// TIA Portal V17 export
// export: Created 2025-03-07T09:17:35.5301543Z, ExportSetting WithDefaults, DisplayName Totally Integrated Automation Portal, DisplayVersion V17 Update 8, DisplayName TIA Portal Openness, DisplayVersion V17 Update 8, DisplayName TIA Portal Version Control Interface, DisplayVersion V17, DisplayName SINAMICS Startdrive Advanced, DisplayVersion V17 SP2, DisplayName SINAMICS Startdrive G110M, G120, G120C, G120D, G120P, G115D, DisplayVersion V17 SP2, DisplayName SINAMICS Startdrive G130, G150, S120, S150, SINAMICS MV, S210, DisplayVersion V17 SP2, DisplayName STEP 7 Professional, DisplayVersion V17 Update 8, DisplayName SINUMERIK ONE STEP 7 Toolbox, DisplayVersion V17 Update 12, DisplayName SINUMERIK 840D sl STEP 7 Toolbox, DisplayVersion V17 Update 12, DisplayName STEP 7 Safety, DisplayVersion V17 Update 6, DisplayName WinCC Advanced, DisplayVersion V17 Update 8
DATA_BLOCK "DB428_OPERATOR_HELP"   // DB428
{ S7_Optimized_Access := 'FALSE' }
VERSION : 1.0
// stored: AutoNumber false, DBAccessibleFromOPCUA true, DBAccessibleFromWebserver true, IsOnlyStoredInLoadMemory false, IsWriteProtectedInAS false
   VAR RETAIN
      HELP_OPERATOR_0 : Bool;   // EMPTY
      HELP_OPERATOR_1 : Bool;   // EMPTY
      HELP_OPERATOR_2 : Bool;   // SPINDLE, POWER MODULE NOT READY
      HELP_OPERATOR_3 : Bool;   // AXIS X, POWER MODULE NOT READY
      HELP_OPERATOR_4 : Bool;   // AXIS Y, POWER MODULE NOT READY
      HELP_OPERATOR_5 : Bool;   // AXIS Z, POWER MODULE NOT READY
      HELP_OPERATOR_6 : Bool;   // AXIS Q, POWER MODULE NOT READY
      HELP_OPERATOR_7 : Bool;   // AXIS A, POWER MODULE NOT READY
      HELP_OPERATOR_8 : Bool;   // AXIS B, POWER MODULE NOT READY
      HELP_OPERATOR_9 : Bool;   // AXIS W, POWER MODULE NOT READY
      HELP_OPERATOR_10 : Bool;   // AXIS E, POWER MODULE NOT READY
      HELP_OPERATOR_11 : Bool;   // AXIS U, POWER MODULE NOT READY
      HELP_OPERATOR_12 : Bool;   // AXIS V, POWER MODULE NOT READY
      HELP_OPERATOR_13 : Bool;   // AXIS ROLLER, POWER MODULE NOT READY
      HELP_OPERATOR_14 : Bool;   // AXIS C, POWER MODULE NOT READY
      HELP_OPERATOR_15 : Bool;   // AXIS DR, POWER MODULE NOT READY
      HELP_OPERATOR_16 : Bool;
      HELP_OPERATOR_17 : Bool;
      HELP_OPERATOR_18 : Bool;
      HELP_OPERATOR_19 : Bool;
      HELP_OPERATOR_20 : Bool;
      HELP_OPERATOR_21 : Bool;
      HELP_OPERATOR_22 : Bool;
      HELP_OPERATOR_23 : Bool;
      HELP_OPERATOR_24 : Bool;
      HELP_OPERATOR_25 : Bool;   // SP11, SPEED NOT 0
      HELP_OPERATOR_26 : Bool;   // SP12, SPEED NOT 0
      HELP_OPERATOR_27 : Bool;   // SP13, SPEED NOT 0
      HELP_OPERATOR_28 : Bool;   // SP14, SPEED NOT 0
      HELP_OPERATOR_29 : Bool;
      HELP_OPERATOR_30 : Bool;
      HELP_OPERATOR_31 : Bool;
      HELP_OPERATOR_32 : Bool;
      HELP_OPERATOR_33 : Bool;   // SP21, SPEED NOT 0
      HELP_OPERATOR_34 : Bool;   // SP22, SPEED NOT 0
      HELP_OPERATOR_35 : Bool;   // SP23, SPEED NOT 0
      HELP_OPERATOR_36 : Bool;   // SP24, SPEED NOT 0
      HELP_OPERATOR_37 : Bool;
      HELP_OPERATOR_38 : Bool;   // RETURN AXIS E10 TO HOME POSITION
      HELP_OPERATOR_39 : Bool;   // RETURN AXIS X13 TO HOME POSITION
      HELP_OPERATOR_40 : Bool;   // RETURN AXIS W11 TO HOME POSITION
      HELP_OPERATOR_41 : Bool;   // RETURN AXIS Z13 TO HOME POSITION
      HELP_OPERATOR_42 : Bool;   // RETURN AXIS E20 TO HOME POSITION
      HELP_OPERATOR_43 : Bool;   // RETURN AXIS C22 TO HOME POSITION
      HELP_OPERATOR_44 : Bool;   // RETURN AXIS X23 TO HOME POSITION
      HELP_OPERATOR_45 : Bool;   // RETURN AXIS W21 TO HOME POSITION
      HELP_OPERATOR_46 : Bool;   // RETURN AXIS Z23 TO HOME POSITION
      HELP_OPERATOR_47 : Bool;   // RETURN AXIS C31 TO HOME POSITION
      HELP_OPERATOR_48 : Bool;
      HELP_OPERATOR_49 : Bool;   // RETURN AXIS X21 TO HOME POSITION
      HELP_OPERATOR_50 : Bool;   // RETURN AXIS Y21 TO HOME POSITION
      HELP_OPERATOR_51 : Bool;   // RETURN AXIS Z21 TO HOME POSITION
      HELP_OPERATOR_52 : Bool;   // RETURN AXIS Z22 TO HOME POSITION
      HELP_OPERATOR_53 : Bool;   // RETURN AXIS Z23 TO HOME POSITION
      HELP_OPERATOR_54 : Bool;   // RETURN AXIS Q21 TO HOME POSITION
      HELP_OPERATOR_55 : Bool;
      HELP_OPERATOR_56 : Bool;
      HELP_OPERATOR_57 : Bool;   // RETURN AXIS B TO HOME POSITION
      HELP_OPERATOR_58 : Bool;   // RETURN AXIS W TO HOME POSITION
      HELP_OPERATOR_59 : Bool;   // RETURN AXIS E TO HOME POSITION
      HELP_OPERATOR_60 : Bool;
      HELP_OPERATOR_61 : Bool;   // RETURN AXIS ROLLER TO HOME POSITION
      HELP_OPERATOR_62 : Bool;   // RETURN AXIS A11 TO HOME POSITION
      HELP_OPERATOR_63 : Bool;   // RETURN AXIS A12 TO HOME POSITION
      HELP_OPERATOR_64 : Bool;   // RETURN AXIS A13 TO HOME POSITION
      HELP_OPERATOR_65 : Bool;   // RETURN AXIS V11 TO HOME POSITION
      HELP_OPERATOR_66 : Bool;   // RETURN AXIS V12 TO HOME POSITION
      HELP_OPERATOR_67 : Bool;   // RETURN AXIS U11 TO HOME POSITION
      HELP_OPERATOR_68 : Bool;   // RETURN AXIS U12 TO HOME POSITION
      HELP_OPERATOR_69 : Bool;   // RETURN AXIS W11 TO HOME POSITION
      HELP_OPERATOR_70 : Bool;   // RETURN AXIS C TO HOME POSITION
      HELP_OPERATOR_71 : Bool;
      HELP_OPERATOR_72 : Bool;   // RETURN AXIS A21 TO HOME POSITION
      HELP_OPERATOR_73 : Bool;   // RETURN AXIS A22 TO HOME POSITION
      HELP_OPERATOR_74 : Bool;   // RETURN AXIS V21 TO HOME POSITION
      HELP_OPERATOR_75 : Bool;
      HELP_OPERATOR_76 : Bool;   // RETURN AXIS U21 TO HOME POSITION
      HELP_OPERATOR_77 : Bool;
      HELP_OPERATOR_78 : Bool;
      HELP_OPERATOR_79 : Bool;   // RETURN AXIS DR1 TO HOME POSITION
      HELP_OPERATOR_80 : Bool;   // RETURN AXIS DR2 TO HOME POSITION
      HELP_OPERATOR_81 : Bool;
      HELP_OPERATOR_82 : Bool;
      HELP_OPERATOR_83 : Bool;   // RETURN AXIS E10 TO OUT OF COLLISION POSITION
      HELP_OPERATOR_84 : Bool;   // RETURN AXIS X13 TO OUT OF COLLISION POSITION
      HELP_OPERATOR_85 : Bool;   // RETURN AXIS W11 TO OUT OF COLLISION POSITION
      HELP_OPERATOR_86 : Bool;   // RETURN AXIS Z13 TO OUT OF COLLISION POSITION
      HELP_OPERATOR_87 : Bool;   // RETURN AXIS E20 TO OUT OF COLLISION POSITION
      HELP_OPERATOR_88 : Bool;   // RETURN AXIS C22 TO OUT OF COLLISION POSITION
      HELP_OPERATOR_89 : Bool;   // RETURN AXIS X23 TO OUT OF COLLISION POSITION
      HELP_OPERATOR_90 : Bool;   // RETURN AXIS W21 TO OUT OF COLLISION POSITION
      HELP_OPERATOR_91 : Bool;   // RETURN AXIS Z23 TO OUT OF COLLISION POSITION
      HELP_OPERATOR_92 : Bool;   // RETURN AXIS C31 TO OUT OF COLLISION POSITION
      HELP_OPERATOR_93 : Bool;   // RETURN AXIS Z23 TO OUT OF COLLISION POSITION
      HELP_OPERATOR_94 : Bool;   // RETURN AXIS Q21 TO OUT OF COLLISION POSITION
      HELP_OPERATOR_95 : Bool;   // RETURN AXIS B TO OUT OF COLLISION POSITION
      HELP_OPERATOR_96 : Bool;   // RETURN AXIS W TO OUT OF COLLISION POSITION
      HELP_OPERATOR_97 : Bool;   // RETURN AXIS E TO OUT OF COLLISION POSITION
      HELP_OPERATOR_98 : Bool;
      HELP_OPERATOR_99 : Bool;   // RETURN AXIS ROLLER TO OUT OF COLLISION POSITION
      HELP_OPERATOR_100 : Bool;   // RETURN AXIS A11 TO OUT OF COLLISION POSITION
      HELP_OPERATOR_101 : Bool;   // RETURN AXIS A12 TO OUT OF COLLISION POSITION
      HELP_OPERATOR_102 : Bool;   // RETURN AXIS A13 TO OUT OF COLLISION POSITION
      HELP_OPERATOR_103 : Bool;   // RETURN AXIS V11 TO OUT OF COLLISION POSITION
      HELP_OPERATOR_104 : Bool;   // RETURN AXIS V12 TO OUT OF COLLISION POSITION
      HELP_OPERATOR_105 : Bool;   // RETURN AXIS U11 TO OUT OF COLLISION POSITION
      HELP_OPERATOR_106 : Bool;   // RETURN AXIS U12 TO OUT OF COLLISION POSITION
      HELP_OPERATOR_107 : Bool;   // RETURN AXIS W11 TO OUT OF COLLISION POSITION
      HELP_OPERATOR_108 : Bool;   // RETURN AXIS C TO OUT OF COLLISION POSITION
      HELP_OPERATOR_109 : Bool;
      HELP_OPERATOR_110 : Bool;   // RETURN AXIS A21 TO OUT OF COLLISION POSITION
      HELP_OPERATOR_111 : Bool;   // RETURN AXIS A22 TO OUT OF COLLISION POSITION
      HELP_OPERATOR_112 : Bool;   // RETURN AXIS V21 TO OUT OF COLLISION POSITION
      HELP_OPERATOR_113 : Bool;
      HELP_OPERATOR_114 : Bool;   // RETURN AXIS U21 TO OUT OF COLLISION POSITION
      HELP_OPERATOR_115 : Bool;
      HELP_OPERATOR_116 : Bool;   // RETURN AXIS DR1 TO OUT OF COLLISION POSITION
      HELP_OPERATOR_117 : Bool;   // RETURN AXIS DR2 TO OUT OF COLLISION POSITION
      HELP_OPERATOR_118 : Bool;
      HELP_OPERATOR_119 : Bool;   // AXIS B NOT IN -180º
      HELP_OPERATOR_120 : Bool;   // AXIS B NOT IN 0º
      HELP_OPERATOR_121 : Bool;   // ROTATE AXIS B TO ANY INDEXING POSITION
      HELP_OPERATOR_122 : Bool;
      HELP_OPERATOR_123 : Bool;
      HELP_OPERATOR_124 : Bool;   // AXIS NOT IN 90º
      HELP_OPERATOR_125 : Bool;   // AXIS NOT IN -90º
      HELP_OPERATOR_126 : Bool;
      HELP_OPERATOR_127 : Bool;
      HELP_OPERATOR_128 : Bool;   // ROTATE AXIS E TO 0º
      HELP_OPERATOR_129 : Bool;   // ROTATE AXIS E TO 180º
      HELP_OPERATOR_130 : Bool;
      HELP_OPERATOR_131 : Bool;
      HELP_OPERATOR_132 : Bool;   // ADVANCE AXIS A
      HELP_OPERATOR_133 : Bool;   // RETURN AXIS A
      HELP_OPERATOR_134 : Bool;   // MOVE AXIS A TO LOAD UNLOAD POSITION
      HELP_OPERATOR_135 : Bool;
      HELP_OPERATOR_136 : Bool;   // ADVANCE AXIS U
      HELP_OPERATOR_137 : Bool;   // RETURN AXIS U
      HELP_OPERATOR_138 : Bool;
      HELP_OPERATOR_139 : Bool;   // RETURN AXIS Q TO POSITION
      HELP_OPERATOR_140 : Bool;
      HELP_OPERATOR_141 : Bool;   // CHOOSE AXES TO ALIGN
      HELP_OPERATOR_142 : Bool;
      HELP_OPERATOR_143 : Bool;
      HELP_OPERATOR_144 : Bool;
      HELP_OPERATOR_145 : Bool;   // ADVANCE AXIS W11
      HELP_OPERATOR_146 : Bool;   // RETURN AXIS W11
      HELP_OPERATOR_147 : Bool;
      HELP_OPERATOR_148 : Bool;
      HELP_OPERATOR_149 : Bool;
      HELP_OPERATOR_150 : Bool;   // RETURN UNIT 01 TO HOME POSITION
      HELP_OPERATOR_151 : Bool;   // RETURN UNIT 02 TO HOME POSITION
      HELP_OPERATOR_152 : Bool;   // RETURN UNIT 03 TO HOME POSITION
      HELP_OPERATOR_153 : Bool;   // RETURN UNIT 04 TO HOME POSITION
      HELP_OPERATOR_154 : Bool;   // RETURN UNIT 05 TO HOME POSITION
      HELP_OPERATOR_155 : Bool;   // RETURN UNIT 06 TO HOME POSITION
      HELP_OPERATOR_156 : Bool;   // RETURN UNIT 07 TO HOME POSITION
      HELP_OPERATOR_157 : Bool;   // RETURN UNIT 08 TO HOME POSITION
      HELP_OPERATOR_158 : Bool;   // RETURN UNIT 09 TO HOME POSITION
      HELP_OPERATOR_159 : Bool;   // RETURN UNIT 10 TO HOME POSITION
      HELP_OPERATOR_160 : Bool;
      HELP_OPERATOR_161 : Bool;
      HELP_OPERATOR_162 : Bool;   // UNIT 01 IN HOME POSITION
      HELP_OPERATOR_163 : Bool;   // UNIT 02 IN HOME POSITION
      HELP_OPERATOR_164 : Bool;   // UNIT 03 IN HOME POSITION
      HELP_OPERATOR_165 : Bool;   // UNIT 04 IN HOME POSITION
      HELP_OPERATOR_166 : Bool;   // UNIT 5 IN HOME POSITION
      HELP_OPERATOR_167 : Bool;   // UNIT 6 IN HOME POSITION
      HELP_OPERATOR_168 : Bool;   // UNIT 7 IN HOME POSITION
      HELP_OPERATOR_169 : Bool;   // UNIT 8 IN HOME POSITION
      HELP_OPERATOR_170 : Bool;   // UNIT 9 IN HOME POSITION
      HELP_OPERATOR_171 : Bool;   // UNIT 10 IN HOME POSITION
      HELP_OPERATOR_172 : Bool;
      HELP_OPERATOR_173 : Bool;
      HELP_OPERATOR_174 : Bool;   // UNIT 01R SPINDLES NOT STOPPED
      HELP_OPERATOR_175 : Bool;   // UNIT 01L SPINDLES NOT STOPPED
      HELP_OPERATOR_176 : Bool;
      HELP_OPERATOR_177 : Bool;
      HELP_OPERATOR_178 : Bool;   // TOOLS IN MAGAZINE 01R NOT OK
      HELP_OPERATOR_179 : Bool;   // TOOLS IN MAGAZINE 01L NOT OK
      HELP_OPERATOR_180 : Bool;
      HELP_OPERATOR_181 : Bool;
      HELP_OPERATOR_182 : Bool;   // RETURN MACHINE TO HOME POSITION
      HELP_OPERATOR_183 : Bool;   // MACHINE IN HOME POSITION
      HELP_OPERATOR_184 : Bool;   // RETURN PART HANDLING DEVICE TO HOME POSITION
      HELP_OPERATOR_185 : Bool;   // PART HANDLING DEVICE IN HOME POSITION
      HELP_OPERATOR_186 : Bool;   // ADVANCE PHD TO LOAD UNLOAD POS FIXTURE
      HELP_OPERATOR_187 : Bool;
      HELP_OPERATOR_188 : Bool;
      HELP_OPERATOR_189 : Bool;
      HELP_OPERATOR_190 : Bool;   // NO PART AT FEED
      HELP_OPERATOR_191 : Bool;   // PARTS DELIVERY OCCUPIED
      HELP_OPERATOR_192 : Bool;
      HELP_OPERATOR_193 : Bool;
      HELP_OPERATOR_194 : Bool;
      HELP_OPERATOR_195 : Bool;
      HELP_OPERATOR_196 : Bool;
      HELP_OPERATOR_197 : Bool;
      HELP_OPERATOR_198 : Bool;
      HELP_OPERATOR_199 : Bool;
      HELP_OPERATOR_200 : Bool;   // SELECT MANUAL MODE
      HELP_OPERATOR_201 : Bool;   // SELECT JOG MODE
      HELP_OPERATOR_202 : Bool;   // SELECT SEMIAUTOMATIC MODE
      HELP_OPERATOR_203 : Bool;   // SELECT TOOL CHANGE MODE
      HELP_OPERATOR_204 : Bool;   // SELECT AUTOMATIC MODE
      HELP_OPERATOR_205 : Bool;   // SELECT INCREMENTAL MODE
      HELP_OPERATOR_206 : Bool;   // SELECT AUTO. OR SEMIAUTO. OR SINGLE MODE
      HELP_OPERATOR_207 : Bool;   // SELECT CALIBRATION CYCLE
      HELP_OPERATOR_208 : Bool;   // SELECT MEASUREMENT CYCLE
      HELP_OPERATOR_209 : Bool;
      HELP_OPERATOR_210 : Bool;
      HELP_OPERATOR_211 : Bool;
      HELP_OPERATOR_212 : Bool;
      HELP_OPERATOR_213 : Bool;
      HELP_OPERATOR_214 : Bool;
      HELP_OPERATOR_215 : Bool;   // UNSELECT REFERENCE MODE
      HELP_OPERATOR_216 : Bool;   // UNSELECT STEP BY STEP MODE
      HELP_OPERATOR_217 : Bool;   // UNSELECT MANUAL LOADING CYCLE
      HELP_OPERATOR_218 : Bool;   // UNSELECT MDA MODE
      HELP_OPERATOR_219 : Bool;   // UNSELECT RUN-OUT CYCLE
      HELP_OPERATOR_220 : Bool;   // UNSELECT DRY CYCLE
      HELP_OPERATOR_221 : Bool;   // UNSELECT GANTRY TEST CYCLE
      HELP_OPERATOR_222 : Bool;   // UNSELECT ROBOT DRY CYCLE
      HELP_OPERATOR_223 : Bool;   // UNSELECT SINGLE CYCLE
      HELP_OPERATOR_224 : Bool;   // UNSELECT CALIBRATION CYCLE
      HELP_OPERATOR_225 : Bool;
      HELP_OPERATOR_226 : Bool;
      HELP_OPERATOR_227 : Bool;
      HELP_OPERATOR_228 : Bool;
      HELP_OPERATOR_229 : Bool;
      HELP_OPERATOR_230 : Bool;   // ENABLE BA1 MODE
      HELP_OPERATOR_231 : Bool;   // ENABLE BA1 OR BA3 MODE
      HELP_OPERATOR_232 : Bool;   // ENABLE BA2 MODE OR CLOSE SAFETY DOORS
      HELP_OPERATOR_233 : Bool;
      HELP_OPERATOR_234 : Bool;
      HELP_OPERATOR_235 : Bool;
      HELP_OPERATOR_236 : Bool;   // SELECT POWDER PLC AUTO MODE
      HELP_OPERATOR_237 : Bool;
      HELP_OPERATOR_238 : Bool;
      HELP_OPERATOR_239 : Bool;
      HELP_OPERATOR_240 : Bool;
      HELP_OPERATOR_241 : Bool;
      HELP_OPERATOR_242 : Bool;
      HELP_OPERATOR_243 : Bool;
      HELP_OPERATOR_244 : Bool;
      HELP_OPERATOR_245 : Bool;
      HELP_OPERATOR_246 : Bool;
      HELP_OPERATOR_247 : Bool;
      HELP_OPERATOR_248 : Bool;
      HELP_OPERATOR_249 : Bool;
      HELP_OPERATOR_250 : Bool;   // OVERRIDE 0
      HELP_OPERATOR_251 : Bool;
      HELP_OPERATOR_252 : Bool;   // EMPTY THE MACHINE
      HELP_OPERATOR_253 : Bool;   // CLEAN GUIDES CYCLE REQUIRED
      HELP_OPERATOR_254 : Bool;   // DISABLE SAVE ENERGY
      HELP_OPERATOR_255 : Bool;   // EMPTY THE CELL
      HELP_OPERATOR_256 : Bool;   // SELECT MANUAL LOADING SELECTOR BUTTON
      HELP_OPERATOR_257 : Bool;
      HELP_OPERATOR_258 : Bool;   // RFID DATA CARRIER CODE MISSING
      HELP_OPERATOR_259 : Bool;   // READING IN PROCESS
      HELP_OPERATOR_260 : Bool;   // WRITING NOT IN PROCESS
      HELP_OPERATOR_261 : Bool;
      HELP_OPERATOR_262 : Bool;
      HELP_OPERATOR_263 : Bool;   // ACKNOWLEDGE QUALITY CHECK
      HELP_OPERATOR_264 : Bool;   // ACKNOWLEDGE ON DEMAND QUALITY CHECK
      HELP_OPERATOR_265 : Bool;   // ACKNOWLEDGE TOOL CHANGED QUALITY CHECK
      HELP_OPERATOR_266 : Bool;   // ACKNOWLEDGE PART TYPE CHANGED QUALITY CHECK
      HELP_OPERATOR_267 : Bool;   // ACKNOWLEDGE FIRST PART QUALITY CHECK
      HELP_OPERATOR_268 : Bool;   // ACKNOWLEDGE CYCLE INTERRUPTED QUALITY CHECK
      HELP_OPERATOR_269 : Bool;   // STOP ACTUAL CYCLE
      HELP_OPERATOR_270 : Bool;   // MACHINE SEQUENCE IN PROGRESS
      HELP_OPERATOR_271 : Bool;   // TEST STOP SEQUENCE IN PROGRESS
      HELP_OPERATOR_272 : Bool;   // SEQUENCE IN PROGRESS
      HELP_OPERATOR_273 : Bool;
      HELP_OPERATOR_274 : Bool;   // LASER FAULT
      HELP_OPERATOR_275 : Bool;   // LASER IS NOT ACTIVE
      HELP_OPERATOR_276 : Bool;   // LASER DEVICE IS NOT READY
      HELP_OPERATOR_277 : Bool;   // LASER EXTERNAL CONTROL IS NOT READY
      HELP_OPERATOR_278 : Bool;   // LASER POINTER FAULT
      HELP_OPERATOR_279 : Bool;
      HELP_OPERATOR_280 : Bool;   // START POWDER UNIT 01
      HELP_OPERATOR_281 : Bool;   // START POWDER UNIT 02
      HELP_OPERATOR_282 : Bool;
      HELP_OPERATOR_283 : Bool;
      HELP_OPERATOR_284 : Bool;
      HELP_OPERATOR_285 : Bool;
      HELP_OPERATOR_286 : Bool;
      HELP_OPERATOR_287 : Bool;
      HELP_OPERATOR_288 : Bool;
      HELP_OPERATOR_289 : Bool;
      HELP_OPERATOR_290 : Bool;   // ACTION ALREADY DONE
      HELP_OPERATOR_291 : Bool;
      HELP_OPERATOR_292 : Bool;
      HELP_OPERATOR_293 : Bool;
      HELP_OPERATOR_294 : Bool;   // JOG MINUS IS NOT ALLOWED
      HELP_OPERATOR_295 : Bool;   // JOG PLUS IS NOT ALLOWED
      HELP_OPERATOR_296 : Bool;
      HELP_OPERATOR_297 : Bool;
      HELP_OPERATOR_298 : Bool;
      HELP_OPERATOR_299 : Bool;
      HELP_OPERATOR_300 : Bool;   // SAFETY GATES NOT CLOSED AND LOCKED
      HELP_OPERATOR_301 : Bool;   // CLOSE AND LOCK MACHINING STATION SAFETY DOOR
      HELP_OPERATOR_302 : Bool;   // OPEN AND UNLOCK MACHINING STATION SAFETY DOOR
      HELP_OPERATOR_303 : Bool;   // CLOSE AND LOCK LOAD/ UNLOAD STATION SAFETY DOOR
      HELP_OPERATOR_304 : Bool;   // OPEN AND UNLOCK LOAD UNLOAD STATION SAFETY DOOR
      HELP_OPERATOR_305 : Bool;   // CLOSE AND LOCK PART HANDLING DEVICE SAFETY DOOR
      HELP_OPERATOR_306 : Bool;   // OPEN AND UNLOCK PART HANDLING DEVICE SAFETY DOOR
      HELP_OPERATOR_307 : Bool;
      HELP_OPERATOR_308 : Bool;   // BIMANUAL NOT PRESSED
      HELP_OPERATOR_309 : Bool;
      HELP_OPERATOR_310 : Bool;
      HELP_OPERATOR_311 : Bool;   // CLOSE AND LOCK TOOL MAGAZINE 01 R SAFETY DOOR
      HELP_OPERATOR_312 : Bool;   // OPEN AND UNLOCK TOOL MAGAZINE 01R SAFETY DOOR
      HELP_OPERATOR_313 : Bool;   // CLOSE AND LOCK TOOL MAGAZINE 01L SAFETY DOOR
      HELP_OPERATOR_314 : Bool;   // OPEN AND UNLOCK TOOL MAGAZINE 01L SAFETY DOOR
      HELP_OPERATOR_315 : Bool;
      HELP_OPERATOR_316 : Bool;
      HELP_OPERATOR_317 : Bool;   // CLOSE AND LOCK UNIT 01 R SAFETY DOOR
      HELP_OPERATOR_318 : Bool;   // OPEN AND UNLOCK UNIT 01R SAFETY DOOR
      HELP_OPERATOR_319 : Bool;   // CLOSE AND LOCK UNIT 01L SAFETY DOOR
      HELP_OPERATOR_320 : Bool;   // OPEN AND UNLOCK UNIT 01L SAFETY DOOR
      HELP_OPERATOR_321 : Bool;
      HELP_OPERATOR_322 : Bool;
      HELP_OPERATOR_323 : Bool;
      HELP_OPERATOR_324 : Bool;
      HELP_OPERATOR_325 : Bool;   // CLOSE AND LOCK MAINTENANCE PLATFORM SAFETY DOOR
      HELP_OPERATOR_326 : Bool;   // OPEN AND UNLOCK MAINTENANCE PLATFORM SAFETY DOOR
      HELP_OPERATOR_327 : Bool;
      HELP_OPERATOR_328 : Bool;
      HELP_OPERATOR_329 : Bool;   // CLOSE AND LOCK CHIP CRUSHER SAFETY DOOR
      HELP_OPERATOR_330 : Bool;   // OPEN AND UNLOCK CHIP CRUSHER SAFETY DOOR
      HELP_OPERATOR_331 : Bool;
      HELP_OPERATOR_332 : Bool;
      HELP_OPERATOR_333 : Bool;   // CLOSE MACHINING STATION SAFETY DOOR
      HELP_OPERATOR_334 : Bool;   // CLOSE LOAD UNLOAD STATION SAFETY DOOR
      HELP_OPERATOR_335 : Bool;   // CLOSE PART HANDLING DEVICE SAFETY DOOR
      HELP_OPERATOR_336 : Bool;
      HELP_OPERATOR_337 : Bool;
      HELP_OPERATOR_338 : Bool;   // CLOSE TOOL MAGAZINE 01R SAFETY DOOR
      HELP_OPERATOR_339 : Bool;   // CLOSE TOOL MAGAZINE 01L SAFETY DOOR
      HELP_OPERATOR_340 : Bool;
      HELP_OPERATOR_341 : Bool;   // CLOSE UNIT 01R SAFETY DOOR
      HELP_OPERATOR_342 : Bool;   // CLOSE UNIT 01L SAFETY DOOR
      HELP_OPERATOR_343 : Bool;
      HELP_OPERATOR_344 : Bool;
      HELP_OPERATOR_345 : Bool;   // CLOSE MAINTENANCE PLATFORM SAFETY DOOR
      HELP_OPERATOR_346 : Bool;
      HELP_OPERATOR_347 : Bool;   // CLOSE CHIP CRUSHER SAFETY DOOR
      HELP_OPERATOR_348 : Bool;
      HELP_OPERATOR_349 : Bool;
      HELP_OPERATOR_350 : Bool;   // PART TYPE 1 SELECTED
      HELP_OPERATOR_351 : Bool;   // PART TYPE 2 SELECTED
      HELP_OPERATOR_352 : Bool;   // PART TYPE 3 SELECTED
      HELP_OPERATOR_353 : Bool;   // PART TYPE 4 SELECTED
      HELP_OPERATOR_354 : Bool;   // PART TYPE 5 SELECTED
      HELP_OPERATOR_355 : Bool;   // PART TYPE 6 SELECTED
      HELP_OPERATOR_356 : Bool;   // PART TYPE 7 SELECTED
      HELP_OPERATOR_357 : Bool;   // PART TYPE 8 SELECTED
      HELP_OPERATOR_358 : Bool;   // PART TYPE 9 SELECTED
      HELP_OPERATOR_359 : Bool;   // PART TYPE 10 SELECTED
      HELP_OPERATOR_360 : Bool;   // PART TYPE 11 SELECTED
      HELP_OPERATOR_361 : Bool;   // PART TYPE 12 SELECTED
      HELP_OPERATOR_362 : Bool;   // PART TYPE 13 SELECTED
      HELP_OPERATOR_363 : Bool;   // PART TYPE 14 SELECTED
      HELP_OPERATOR_364 : Bool;   // PART TYPE 15 SELECTED
      HELP_OPERATOR_365 : Bool;   // PART TYPE 16 SELECTED
      HELP_OPERATOR_366 : Bool;   // PART TYPE 17 SELECTED
      HELP_OPERATOR_367 : Bool;   // PART TYPE 18 SELECTED
      HELP_OPERATOR_368 : Bool;   // PART TYPE 19 SELECTED
      HELP_OPERATOR_369 : Bool;   // PART TYPE 20 SELECTED
      HELP_OPERATOR_370 : Bool;   // PART TYPE 21 SELECTED
      HELP_OPERATOR_371 : Bool;   // PART TYPE 22 SELECTED
      HELP_OPERATOR_372 : Bool;   // PART TYPE 23 SELECTED
      HELP_OPERATOR_373 : Bool;   // PART TYPE 24 SELECTED
      HELP_OPERATOR_374 : Bool;   // PART TYPE 25 SELECTED
      HELP_OPERATOR_375 : Bool;   // PART TYPE 26 SELECTED
      HELP_OPERATOR_376 : Bool;   // PART TYPE 27 SELECTED
      HELP_OPERATOR_377 : Bool;   // PART TYPE 28 SELECTED
      HELP_OPERATOR_378 : Bool;   // PART TYPE 29 SELECTED
      HELP_OPERATOR_379 : Bool;   // PART TYPE 30 SELECTED
      HELP_OPERATOR_380 : Bool;   // PART TYPE 31 SELECTED
      HELP_OPERATOR_381 : Bool;   // PART TYPE 32 SELECTED
      HELP_OPERATOR_382 : Bool;
      HELP_OPERATOR_383 : Bool;
      HELP_OPERATOR_384 : Bool;
      HELP_OPERATOR_385 : Bool;
      HELP_OPERATOR_386 : Bool;
      HELP_OPERATOR_387 : Bool;
      HELP_OPERATOR_388 : Bool;
      HELP_OPERATOR_389 : Bool;
      HELP_OPERATOR_390 : Bool;
      HELP_OPERATOR_391 : Bool;
      HELP_OPERATOR_392 : Bool;
      HELP_OPERATOR_393 : Bool;
      HELP_OPERATOR_394 : Bool;
      HELP_OPERATOR_395 : Bool;
      HELP_OPERATOR_396 : Bool;
      HELP_OPERATOR_397 : Bool;
      HELP_OPERATOR_398 : Bool;
      HELP_OPERATOR_399 : Bool;
      HELP_OPERATOR_400 : Bool;   // CONFIRM HARDWARE DISABLING
      HELP_OPERATOR_401 : Bool;
      HELP_OPERATOR_402 : Bool;   // PART A DISABLED
      HELP_OPERATOR_403 : Bool;   // PART B DISABLED
      HELP_OPERATOR_404 : Bool;   // PART C DISABLED
      HELP_OPERATOR_405 : Bool;   // PART D DISABLED
      HELP_OPERATOR_406 : Bool;
      HELP_OPERATOR_407 : Bool;
      HELP_OPERATOR_408 : Bool;
      HELP_OPERATOR_409 : Bool;
      HELP_OPERATOR_410 : Bool;   // FIXTURE 1 DISABLED
      HELP_OPERATOR_411 : Bool;   // FIXTURE 2 DISABLED
      HELP_OPERATOR_412 : Bool;
      HELP_OPERATOR_413 : Bool;
      HELP_OPERATOR_414 : Bool;   // UNIT 01 DISABLED
      HELP_OPERATOR_415 : Bool;   // UNIT 02 DISABLED
      HELP_OPERATOR_416 : Bool;   // UNIT 03 DISABLED
      HELP_OPERATOR_417 : Bool;
      HELP_OPERATOR_418 : Bool;
      HELP_OPERATOR_419 : Bool;   // ALL BK MIKRO 01R UNITS DISABLED
      HELP_OPERATOR_420 : Bool;   // ALL BK MIKRO 01L UNITS DISABLED
      HELP_OPERATOR_421 : Bool;
      HELP_OPERATOR_422 : Bool;
      HELP_OPERATOR_423 : Bool;
      HELP_OPERATOR_424 : Bool;   // LASER SOURCE DISABLED
      HELP_OPERATOR_425 : Bool;
      HELP_OPERATOR_426 : Bool;
      HELP_OPERATOR_427 : Bool;
      HELP_OPERATOR_428 : Bool;
      HELP_OPERATOR_429 : Bool;
      HELP_OPERATOR_430 : Bool;
      HELP_OPERATOR_431 : Bool;
      HELP_OPERATOR_432 : Bool;
      HELP_OPERATOR_433 : Bool;
      HELP_OPERATOR_434 : Bool;
      HELP_OPERATOR_435 : Bool;
      HELP_OPERATOR_436 : Bool;
      HELP_OPERATOR_437 : Bool;
      HELP_OPERATOR_438 : Bool;
      HELP_OPERATOR_439 : Bool;
      HELP_OPERATOR_440 : Bool;   // PHD ARM 1, PART PRESENT
      HELP_OPERATOR_441 : Bool;   // PHD ARM 2, PART PRESENT
      HELP_OPERATOR_442 : Bool;
      HELP_OPERATOR_443 : Bool;
      HELP_OPERATOR_444 : Bool;   // NO PART PRESENT
      HELP_OPERATOR_445 : Bool;   // NO MASTER PART PRESENT
      HELP_OPERATOR_446 : Bool;   // FIXTURE IN UNIT 01 CLADDING STATION NOT CLAMPED
      HELP_OPERATOR_447 : Bool;
      HELP_OPERATOR_448 : Bool;
      HELP_OPERATOR_449 : Bool;
      HELP_OPERATOR_450 : Bool;
      HELP_OPERATOR_451 : Bool;
      HELP_OPERATOR_452 : Bool;
      HELP_OPERATOR_453 : Bool;
      HELP_OPERATOR_454 : Bool;
      HELP_OPERATOR_455 : Bool;
      HELP_OPERATOR_456 : Bool;
      HELP_OPERATOR_457 : Bool;
      HELP_OPERATOR_458 : Bool;
      HELP_OPERATOR_459 : Bool;
      HELP_OPERATOR_460 : Bool;   // SP11, TOOL CLAMPING CLAMPED WITHOUT TOOL
      HELP_OPERATOR_461 : Bool;   // SP12, TOOL CLAMPING CLAMPED WITHOUT TOOL
      HELP_OPERATOR_462 : Bool;   // SP13, TOOL CLAMPING CLAMPED WITHOUT TOOL
      HELP_OPERATOR_463 : Bool;   // SP14, TOOL CLAMPING CLAMPED WITHOUT TOOL
      HELP_OPERATOR_464 : Bool;
      HELP_OPERATOR_465 : Bool;
      HELP_OPERATOR_466 : Bool;   // SP21, TOOL CLAMPING CLAMPED WITHOUT TOOL
      HELP_OPERATOR_467 : Bool;   // SP22, TOOL CLAMPING CLAMPED WITHOUT TOOL
      HELP_OPERATOR_468 : Bool;   // SP23, TOOL CLAMPING CLAMPED WITHOUT TOOL
      HELP_OPERATOR_469 : Bool;   // SP24, TOOL CLAMPING CLAMPED WITHOUT TOOL
      HELP_OPERATOR_470 : Bool;
      HELP_OPERATOR_471 : Bool;
      HELP_OPERATOR_472 : Bool;   // SP11, UNCLAMP TOOL CLAMPING
      HELP_OPERATOR_473 : Bool;   // SP12, UNCLAMP TOOL CLAMPING
      HELP_OPERATOR_474 : Bool;   // SP13, UNCLAMP TOOL CLAMPING
      HELP_OPERATOR_475 : Bool;   // SP14, UNCLAMP TOOL CLAMPING
      HELP_OPERATOR_476 : Bool;
      HELP_OPERATOR_477 : Bool;
      HELP_OPERATOR_478 : Bool;   // SP21, UNCLAMP TOOL CLAMPING
      HELP_OPERATOR_479 : Bool;   // SP22, UNCLAMP TOOL CLAMPING
      HELP_OPERATOR_480 : Bool;   // SP23, UNCLAMP TOOL CLAMPING
      HELP_OPERATOR_481 : Bool;   // SP24, UNCLAMP TOOL CLAMPING
      HELP_OPERATOR_482 : Bool;
      HELP_OPERATOR_483 : Bool;
      HELP_OPERATOR_484 : Bool;   // SP11, CLAMP TOOL CLAMPING
      HELP_OPERATOR_485 : Bool;   // SP12, CLAMP TOOL CLAMPING
      HELP_OPERATOR_486 : Bool;   // SP13, CLAMP TOOL CLAMPING
      HELP_OPERATOR_487 : Bool;   // SP14, CLAMP TOOL CLAMPING
      HELP_OPERATOR_488 : Bool;
      HELP_OPERATOR_489 : Bool;
      HELP_OPERATOR_490 : Bool;   // SP21, CLAMP TOOL CLAMPING
      HELP_OPERATOR_491 : Bool;   // SP22, CLAMP TOOL CLAMPING
      HELP_OPERATOR_492 : Bool;   // SP23, CLAMP TOOL CLAMPING
      HELP_OPERATOR_493 : Bool;   // SP24, CLAMP TOOL CLAMPING
      HELP_OPERATOR_494 : Bool;
      HELP_OPERATOR_495 : Bool;
      HELP_OPERATOR_496 : Bool;   // CLAMP WITH TOOL
      HELP_OPERATOR_497 : Bool;   // CLAMP TOOL CLAMPING
      HELP_OPERATOR_498 : Bool;
      HELP_OPERATOR_499 : Bool;   // MOVE TOOL FROM SP11 TO TOOL MAGAZINE 01R
      HELP_OPERATOR_500 : Bool;   // MOVE TOOL FROM SP12 TO TOOL MAGAZINE 01R
      HELP_OPERATOR_501 : Bool;   // MOVE TOOL FROM SP13 TO TOOL MAGAZINE 01R
      HELP_OPERATOR_502 : Bool;   // MOVE TOOL FROM SP14 TO TOOL MAGAZINE 01R
      HELP_OPERATOR_503 : Bool;
      HELP_OPERATOR_504 : Bool;
      HELP_OPERATOR_505 : Bool;   // MOVE TOOL FROM SP21 TO TOOL MAGAZINE 01L
      HELP_OPERATOR_506 : Bool;   // MOVE TOOL FROM SP22 TO TOOL MAGAZINE 01L
      HELP_OPERATOR_507 : Bool;   // MOVE TOOL FROM SP23 TO TOOL MAGAZINE 01L
      HELP_OPERATOR_508 : Bool;   // MOVE TOOL FROM SP24 TO TOOL MAGAZINE 01L
      HELP_OPERATOR_509 : Bool;
      HELP_OPERATOR_510 : Bool;
      HELP_OPERATOR_511 : Bool;   // SP11, ENABLE TOOL MONITORING
      HELP_OPERATOR_512 : Bool;   // SP12, ENABLE TOOL MONITORING
      HELP_OPERATOR_513 : Bool;   // SP13, ENABLE TOOL MONITORING
      HELP_OPERATOR_514 : Bool;   // SP14, ENABLE TOOL MONITORING
      HELP_OPERATOR_515 : Bool;
      HELP_OPERATOR_516 : Bool;
      HELP_OPERATOR_517 : Bool;   // SP21, ENABLE TOOL MONITORING
      HELP_OPERATOR_518 : Bool;   // SP22, ENABLE TOOL MONITORING
      HELP_OPERATOR_519 : Bool;   // SP23, ENABLE TOOL MONITORING
      HELP_OPERATOR_520 : Bool;   // SP24, ENABLE TOOL MONITORING
      HELP_OPERATOR_521 : Bool;
      HELP_OPERATOR_522 : Bool;
      HELP_OPERATOR_523 : Bool;   // BK MIKRO SP11 SEND TO HOME POS OR DISCONNECT CABLE
      HELP_OPERATOR_524 : Bool;   // BK MIKRO SP12 SEND TO HOME POS OR DISCONNECT CABLE
      HELP_OPERATOR_525 : Bool;   // BK MIKRO SP13 SEND TO HOME POS OR DISCONNECT CABLE
      HELP_OPERATOR_526 : Bool;   // BK MIKRO SP14 SEND TO HOME POS OR DISCONNECT CABLE
      HELP_OPERATOR_527 : Bool;
      HELP_OPERATOR_528 : Bool;
      HELP_OPERATOR_529 : Bool;   // BK MIKRO SP21 SEND TO HOME POS OR DISCONNECT CABLE
      HELP_OPERATOR_530 : Bool;   // BK MIKRO SP22 SEND TO HOME POS OR DISCONNECT CABLE
      HELP_OPERATOR_531 : Bool;   // BK MIKRO SP23 SEND TO HOME POS OR DISCONNECT CABLE
      HELP_OPERATOR_532 : Bool;   // BK MIKRO SP24 SEND TO HOME POS OR DISCONNECT CABLE
      HELP_OPERATOR_533 : Bool;
      HELP_OPERATOR_534 : Bool;
      HELP_OPERATOR_535 : Bool;   // MAIN OPERATOR PANEL, PRESS BUTTON CONTROL ON
      HELP_OPERATOR_536 : Bool;   // MAIN OPERATOR PANEL, PRESS BUTTON RESET
      HELP_OPERATOR_537 : Bool;   // REMOVE EMERGENCY STOPS, PRESS RESET FAULTS
      HELP_OPERATOR_538 : Bool;   // MACHINE STOP SERVICES DELAYED ENABLED
      HELP_OPERATOR_539 : Bool;
      HELP_OPERATOR_540 : Bool;
      HELP_OPERATOR_541 : Bool;   // SWITCH ON HYDRAULIC SYSTEM
      HELP_OPERATOR_542 : Bool;   // SWITCH ON PNEUMATIC SYSTEM
      HELP_OPERATOR_543 : Bool;   // LUBRICATION PRESSURES SWITCHES NOT BELOW 2 BARS
      HELP_OPERATOR_544 : Bool;   // MAIN CHIP CONVEYOR CONTAINER NOT PRESENT
      HELP_OPERATOR_545 : Bool;
      HELP_OPERATOR_546 : Bool;
      HELP_OPERATOR_547 : Bool;   // OPEN COOLANT VALVE
      HELP_OPERATOR_548 : Bool;   // SWITCH ON CHIP CRUSHER
      HELP_OPERATOR_549 : Bool;   // SWITCH OFF CHIP CRUSHER
      HELP_OPERATOR_550 : Bool;
      HELP_OPERATOR_551 : Bool;
      HELP_OPERATOR_552 : Bool;   // FILTER PAPER BAND HIGH LEVEL
      HELP_OPERATOR_553 : Bool;   // NOT READY
      HELP_OPERATOR_554 : Bool;   // LOW LEVEL
      HELP_OPERATOR_555 : Bool;   // NO PRESSURE AT INPUT
      HELP_OPERATOR_556 : Bool;   // FILTER CLOGGED
      HELP_OPERATOR_557 : Bool;
      HELP_OPERATOR_558 : Bool;
      HELP_OPERATOR_559 : Bool;   // FLUSH FILTER 01R NOT IN HOME POSITION
      HELP_OPERATOR_560 : Bool;   // FLUSH FILTER 01L NOT IN HOME POSITION
      HELP_OPERATOR_561 : Bool;
      HELP_OPERATOR_562 : Bool;
      HELP_OPERATOR_563 : Bool;
      HELP_OPERATOR_564 : Bool;
      HELP_OPERATOR_565 : Bool;   // SWITCH ON MQL PUMP
      HELP_OPERATOR_566 : Bool;
      HELP_OPERATOR_567 : Bool;   // SWITCH OFF MQL SP11
      HELP_OPERATOR_568 : Bool;   // SWITCH OFF MQL SP12
      HELP_OPERATOR_569 : Bool;   // SWITCH OFF MQL SP13
      HELP_OPERATOR_570 : Bool;   // SWITCH OFF MQL SP14
      HELP_OPERATOR_571 : Bool;
      HELP_OPERATOR_572 : Bool;
      HELP_OPERATOR_573 : Bool;   // SWITCH OFF MQL SP21
      HELP_OPERATOR_574 : Bool;   // SWITCH OFF MQL SP22
      HELP_OPERATOR_575 : Bool;   // SWITCH OFF MQL SP23
      HELP_OPERATOR_576 : Bool;   // SWITCH OFF MQL SP24
      HELP_OPERATOR_577 : Bool;
      HELP_OPERATOR_578 : Bool;
      HELP_OPERATOR_579 : Bool;
      HELP_OPERATOR_580 : Bool;
      HELP_OPERATOR_581 : Bool;
      HELP_OPERATOR_582 : Bool;
      HELP_OPERATOR_583 : Bool;
      HELP_OPERATOR_584 : Bool;
      HELP_OPERATOR_585 : Bool;
      HELP_OPERATOR_586 : Bool;
      HELP_OPERATOR_587 : Bool;
      HELP_OPERATOR_588 : Bool;
      HELP_OPERATOR_589 : Bool;
      HELP_OPERATOR_590 : Bool;   // CLAMP FIXTURE 1
      HELP_OPERATOR_591 : Bool;   // UNCLAMP FIXTURE 1
      HELP_OPERATOR_592 : Bool;   // CLAMP OR UNCLAMP FIXTURE 1
      HELP_OPERATOR_593 : Bool;   // FIXTURE 1, CLAMPED
      HELP_OPERATOR_594 : Bool;   // FIXTURE 1, UNCLAMPED
      HELP_OPERATOR_595 : Bool;   // SELECT PART TYPE FIXTURE 1
      HELP_OPERATOR_596 : Bool;   // FIXTURE 1 PART NOT OK
      HELP_OPERATOR_597 : Bool;   // CLAMPING SEQUENCE F1 IN PROGRESS
      HELP_OPERATOR_598 : Bool;
      HELP_OPERATOR_599 : Bool;   // CLAMP FIXTURE 2
      HELP_OPERATOR_600 : Bool;   // UNCLAMP FIXTURE 2
      HELP_OPERATOR_601 : Bool;   // CLAMP OR UNCLAMP FIXTURE 2
      HELP_OPERATOR_602 : Bool;   // FIXTURE 2, CLAMPED
      HELP_OPERATOR_603 : Bool;   // FIXTURE 2, UNCLAMPED
      HELP_OPERATOR_604 : Bool;   // SELECT PART TYPE FIXTURE 2
      HELP_OPERATOR_605 : Bool;   // FIXTURE 2 PART NOT OK
      HELP_OPERATOR_606 : Bool;   // CLAMPING SEQUENCE F2 IN PROGRESS
      HELP_OPERATOR_607 : Bool;
      HELP_OPERATOR_608 : Bool;   // CLAMP FIXTURE 3
      HELP_OPERATOR_609 : Bool;   // UNCLAMP FIXTURE 3
      HELP_OPERATOR_610 : Bool;   // CLAMP OR UNCLAMP FIXTURE 3
      HELP_OPERATOR_611 : Bool;   // FIXTURE 3, CLAMPED
      HELP_OPERATOR_612 : Bool;   // FIXTURE 3, UNCLAMPED
      HELP_OPERATOR_613 : Bool;   // SELECT PART TYPE FIXTURE 3
      HELP_OPERATOR_614 : Bool;   // FIXTURE 3 PART NOT OK
      HELP_OPERATOR_615 : Bool;   // CLAMPING SEQUENCE F3 IN PROGRESS
      HELP_OPERATOR_616 : Bool;
      HELP_OPERATOR_617 : Bool;   // CLAMP FIXTURE 4
      HELP_OPERATOR_618 : Bool;   // UNCLAMP FIXTURE 4
      HELP_OPERATOR_619 : Bool;   // CLAMP OR UNCLAMP FIXTURE 4
      HELP_OPERATOR_620 : Bool;   // FIXTURE 4, CLAMPED
      HELP_OPERATOR_621 : Bool;   // FIXTURE 4, UNCLAMPED
      HELP_OPERATOR_622 : Bool;   // SELECT PART TYPE FIXTURE 4
      HELP_OPERATOR_623 : Bool;   // FIXTURE 4 PART NOT OK
      HELP_OPERATOR_624 : Bool;   // CLAMPING SEQUENCE F4 IN PROGRESS
      HELP_OPERATOR_625 : Bool;
      HELP_OPERATOR_626 : Bool;   // LOCATE AXIAL LOCATOR
      HELP_OPERATOR_627 : Bool;   // LOCATE AXIAL LOCATOR CARRIER
      HELP_OPERATOR_628 : Bool;   // LOCATE RADIAL LOCATOR
      HELP_OPERATOR_629 : Bool;   // LOCATE RADIAL LOCATOR CARRIER
      HELP_OPERATOR_630 : Bool;   // CLAMP CLAMPING FLANGE
      HELP_OPERATOR_631 : Bool;   // ADVANCE TAILSTOCK
      HELP_OPERATOR_632 : Bool;   // LOCATE SHIFTING DEVICE
      HELP_OPERATOR_633 : Bool;   // BLOCK BLOCKING DEVICE
      HELP_OPERATOR_634 : Bool;   // CLAMP VIBRATION DAMPER
      HELP_OPERATOR_635 : Bool;   // CLAMP JAW CHUCK
      HELP_OPERATOR_636 : Bool;   // CLAMP CENTRAL JAWCHUCK
      HELP_OPERATOR_637 : Bool;   // CLAMP ROTARY JAW CHUCK
      HELP_OPERATOR_638 : Bool;   // ADVANCE REMOVABLE STOP
      HELP_OPERATOR_639 : Bool;
      HELP_OPERATOR_640 : Bool;
      HELP_OPERATOR_641 : Bool;
      HELP_OPERATOR_642 : Bool;   // CLAMP OR UNCLAMP FIXTURE IN UNIT 01 STATION 1
      HELP_OPERATOR_643 : Bool;   // CLAMP FIXTURE IN UNIT 1 STATION 3
      HELP_OPERATOR_644 : Bool;   // CLAMP FIXTURE IN UNIT 1 STATION 4
      HELP_OPERATOR_645 : Bool;   // CLAMP OR UNCLAMP FIXTURE IN UNIT 02 STATION 1
      HELP_OPERATOR_646 : Bool;   // CLAMP FIXTURE IN UNIT 2 STATION 2
      HELP_OPERATOR_647 : Bool;   // CLAMP FIXTURE IN UNIT 2 STATION 3
      HELP_OPERATOR_648 : Bool;   // CLAMP FIXTURE IN UNIT 2 STATION 4
      HELP_OPERATOR_649 : Bool;
      HELP_OPERATOR_650 : Bool;   // RETURN STATION 1 TO HOME POSITION
      HELP_OPERATOR_651 : Bool;   // RETURN STATION 2 TO HOME POSITION
      HELP_OPERATOR_652 : Bool;   // RETURN STATION 3 TO HOME POSITION
      HELP_OPERATOR_653 : Bool;   // RETURN STATION 4 TO HOME POSITION
      HELP_OPERATOR_654 : Bool;
      HELP_OPERATOR_655 : Bool;
      HELP_OPERATOR_656 : Bool;   // UNIT 01 ALL FIXTURES NOT CLAMPED
      HELP_OPERATOR_657 : Bool;   // UNIT 02 ALL FIXTURES NOT CLAMPED
      HELP_OPERATOR_658 : Bool;
      HELP_OPERATOR_659 : Bool;
      HELP_OPERATOR_660 : Bool;
      HELP_OPERATOR_661 : Bool;
      HELP_OPERATOR_662 : Bool;
      HELP_OPERATOR_663 : Bool;
      HELP_OPERATOR_664 : Bool;   // RETURN AXIAL LOCATOR
      HELP_OPERATOR_665 : Bool;   // RETURN AXIAL LOCATOR CARRIER
      HELP_OPERATOR_666 : Bool;   // RETURN RADIAL LOCATOR
      HELP_OPERATOR_667 : Bool;   // RETURN RADIAL LOCATOR CARRIER
      HELP_OPERATOR_668 : Bool;   // UNCLAMP CLAMPING FLANGE
      HELP_OPERATOR_669 : Bool;   // RETURN TAILSTOCK
      HELP_OPERATOR_670 : Bool;   // RETURN SHIFTING DEVICE
      HELP_OPERATOR_671 : Bool;   // UNBLOCK BLOCKING DEVICE
      HELP_OPERATOR_672 : Bool;   // UNCLAMP VIBRATION DAMPER
      HELP_OPERATOR_673 : Bool;   // UNCLAMP JAW CHUCK
      HELP_OPERATOR_674 : Bool;   // UNCLAMP CENTRAL JAWCHUCK
      HELP_OPERATOR_675 : Bool;   // UNCLAMP ROTARY JAW CHUCK
      HELP_OPERATOR_676 : Bool;   // RETURN REMOVABLE STOP
      HELP_OPERATOR_677 : Bool;
      HELP_OPERATOR_678 : Bool;
      HELP_OPERATOR_679 : Bool;
      HELP_OPERATOR_680 : Bool;   // MACHINE ANY FIXTURE CALIBRATION MISSING
      HELP_OPERATOR_681 : Bool;
      HELP_OPERATOR_682 : Bool;
      HELP_OPERATOR_683 : Bool;
      HELP_OPERATOR_684 : Bool;
      HELP_OPERATOR_685 : Bool;
      HELP_OPERATOR_686 : Bool;
      HELP_OPERATOR_687 : Bool;
      HELP_OPERATOR_688 : Bool;
      HELP_OPERATOR_689 : Bool;
      HELP_OPERATOR_690 : Bool;
      HELP_OPERATOR_691 : Bool;
      HELP_OPERATOR_692 : Bool;
      HELP_OPERATOR_693 : Bool;
      HELP_OPERATOR_694 : Bool;
      HELP_OPERATOR_695 : Bool;
      HELP_OPERATOR_696 : Bool;
      HELP_OPERATOR_697 : Bool;
      HELP_OPERATOR_698 : Bool;
      HELP_OPERATOR_699 : Bool;
      HELP_OPERATOR_700 : Bool;
      HELP_OPERATOR_701 : Bool;
      HELP_OPERATOR_702 : Bool;   // RELIEVE PRESSURE AXIAL LOCATOR
      HELP_OPERATOR_703 : Bool;   // RELIEVE PRESSURE AXIAL LOCATOR CARRIER
      HELP_OPERATOR_704 : Bool;   // RELIEVE PRESSURE RADIAL LOCATOR
      HELP_OPERATOR_705 : Bool;   // RELIEVE PRESSURE RADIAL LOCATOR CARRIER
      HELP_OPERATOR_706 : Bool;   // RELIEVE PRESSURE CLAMPING FLANGE
      HELP_OPERATOR_707 : Bool;   // RELIEVE PRESSURE TAILSTOCK
      HELP_OPERATOR_708 : Bool;   // RELIEVE PRESSURE SHIFTING DEVICE
      HELP_OPERATOR_709 : Bool;   // RELIEVE PRESSURE BLOCKING DEVICE
      HELP_OPERATOR_710 : Bool;   // RELIEVE PRESSURE VIBRATION DAMPER
      HELP_OPERATOR_711 : Bool;   // RELIEVE PRESSURE JAW CHUCK
      HELP_OPERATOR_712 : Bool;   // RELIEVE PRESSURE CENTRAL JAW CHUCK
      HELP_OPERATOR_713 : Bool;   // RELIEVE PRESSURE ROTARY JAW CHUCK
      HELP_OPERATOR_714 : Bool;   // RELIEVE PRESSURE REMOVABLE STOP
      HELP_OPERATOR_715 : Bool;
      HELP_OPERATOR_716 : Bool;
      HELP_OPERATOR_717 : Bool;
      HELP_OPERATOR_718 : Bool;
      HELP_OPERATOR_719 : Bool;
      HELP_OPERATOR_720 : Bool;
      HELP_OPERATOR_721 : Bool;
      HELP_OPERATOR_722 : Bool;
      HELP_OPERATOR_723 : Bool;
      HELP_OPERATOR_724 : Bool;
      HELP_OPERATOR_725 : Bool;
      HELP_OPERATOR_726 : Bool;
      HELP_OPERATOR_727 : Bool;
      HELP_OPERATOR_728 : Bool;
      HELP_OPERATOR_729 : Bool;
      HELP_OPERATOR_730 : Bool;
      HELP_OPERATOR_731 : Bool;
      HELP_OPERATOR_732 : Bool;
      HELP_OPERATOR_733 : Bool;
      HELP_OPERATOR_734 : Bool;
      HELP_OPERATOR_735 : Bool;
      HELP_OPERATOR_736 : Bool;
      HELP_OPERATOR_737 : Bool;
      HELP_OPERATOR_738 : Bool;
      HELP_OPERATOR_739 : Bool;
      HELP_OPERATOR_740 : Bool;   // CLAMP GRIPPER PHD ARM 1
      HELP_OPERATOR_741 : Bool;   // CLAMP GRIPPER A , PHD ARM 1
      HELP_OPERATOR_742 : Bool;   // CLAMP GRIPPER B , PHD ARM 1
      HELP_OPERATOR_743 : Bool;   // CLAMP GRIPPER C , PHD ARM 1
      HELP_OPERATOR_744 : Bool;   // CLAMP GRIPPER D , PHD ARM 1
      HELP_OPERATOR_745 : Bool;   // CLAMP GRIPPER PHD ARM 2
      HELP_OPERATOR_746 : Bool;   // CLAMP GRIPPER A , PHD ARM 2
      HELP_OPERATOR_747 : Bool;   // CLAMP GRIPPER B , PHD ARM 2
      HELP_OPERATOR_748 : Bool;   // CLAMP GRIPPER C , PHD ARM 2
      HELP_OPERATOR_749 : Bool;   // CLAMP GRIPPER D , PHD ARM 2
      HELP_OPERATOR_750 : Bool;
      HELP_OPERATOR_751 : Bool;
      HELP_OPERATOR_752 : Bool;   // UNCLAMP GRIPPER PHD ARM 1
      HELP_OPERATOR_753 : Bool;   // UNCLAMP GRIPPER A , PHD ARM 1
      HELP_OPERATOR_754 : Bool;   // UNCLAMP GRIPPER B , PHD ARM 1
      HELP_OPERATOR_755 : Bool;   // UNCLAMP GRIPPER C , PHD ARM 1
      HELP_OPERATOR_756 : Bool;   // UNCLAMP GRIPPER D , PHD ARM 1
      HELP_OPERATOR_757 : Bool;   // UNCLAMP GRIPPER PHD ARM 2
      HELP_OPERATOR_758 : Bool;   // UNCLAMP GRIPPER A , PHD ARM 2
      HELP_OPERATOR_759 : Bool;   // UNCLAMP GRIPPER B , PHD ARM 2
      HELP_OPERATOR_760 : Bool;   // UNCLAMP GRIPPER C , PHD ARM 2
      HELP_OPERATOR_761 : Bool;   // UNCLAMP GRIPPER D , PHD ARM 2
      HELP_OPERATOR_762 : Bool;
      HELP_OPERATOR_763 : Bool;
      HELP_OPERATOR_764 : Bool;   // RETURN CLEAN TOOL-HOLDER
      HELP_OPERATOR_765 : Bool;   // ADVANCE CLEAN TOOL-HOLDER
      HELP_OPERATOR_766 : Bool;
      HELP_OPERATOR_767 : Bool;
      HELP_OPERATOR_768 : Bool;   // TOOL MAGAZINE RETURN RFID READ/WRITE HEAD CARRIER
      HELP_OPERATOR_769 : Bool;   // TOOL MAGAZINE LOCATE RFID READ/WRITE HEAD CARRIER
      HELP_OPERATOR_770 : Bool;
      HELP_OPERATOR_771 : Bool;
      HELP_OPERATOR_772 : Bool;   // RISE LOAD UNLOAD LIFTING SLIDE
      HELP_OPERATOR_773 : Bool;   // RETURN LOAD UNLOAD LIFTING SLIDE
      HELP_OPERATOR_774 : Bool;
      HELP_OPERATOR_775 : Bool;   // POLE IDENTIFICATION NOT DONE
      HELP_OPERATOR_776 : Bool;   // UNBLOCK TABLE
      HELP_OPERATOR_777 : Bool;   // OPEN HATCH
      HELP_OPERATOR_778 : Bool;   // CLOSE HATCH
      HELP_OPERATOR_779 : Bool;   // OPEN AUTOMATIC DOOR
      HELP_OPERATOR_780 : Bool;
      HELP_OPERATOR_781 : Bool;
      HELP_OPERATOR_782 : Bool;   // UNBLOCK SAFETY BRAKE AXIS Z
      HELP_OPERATOR_783 : Bool;   // UNLOCK AXIS Z MAINTENANCE BRAKE
      HELP_OPERATOR_784 : Bool;   // NOT IN STORED POSITION AXIS Y MAINTENANCE BRAKE
      HELP_OPERATOR_785 : Bool;   // LIFTING SLIDE VERTICAL STOP NOT IN POSITION
      HELP_OPERATOR_786 : Bool;   // ROLLER HOLDING BRAKE NOT OPENED
      HELP_OPERATOR_787 : Bool;
      HELP_OPERATOR_788 : Bool;   // RETURN CYLINDER
      HELP_OPERATOR_789 : Bool;
      HELP_OPERATOR_790 : Bool;
      HELP_OPERATOR_791 : Bool;
      HELP_OPERATOR_792 : Bool;   // OPEN SEALING STRUCTURES
      HELP_OPERATOR_793 : Bool;   // CLOSE SEALING STRUCTURES
      HELP_OPERATOR_794 : Bool;
      HELP_OPERATOR_795 : Bool;
      HELP_OPERATOR_796 : Bool;
      HELP_OPERATOR_797 : Bool;
      HELP_OPERATOR_798 : Bool;
      HELP_OPERATOR_799 : Bool;
      HELP_OPERATOR_800 : Bool;
      HELP_OPERATOR_801 : Bool;
      HELP_OPERATOR_802 : Bool;
      HELP_OPERATOR_803 : Bool;
      HELP_OPERATOR_804 : Bool;
      HELP_OPERATOR_805 : Bool;
      HELP_OPERATOR_806 : Bool;
      HELP_OPERATOR_807 : Bool;
      HELP_OPERATOR_808 : Bool;
      HELP_OPERATOR_809 : Bool;
      HELP_OPERATOR_810 : Bool;
      HELP_OPERATOR_811 : Bool;
      HELP_OPERATOR_812 : Bool;
      HELP_OPERATOR_813 : Bool;
      HELP_OPERATOR_814 : Bool;
      HELP_OPERATOR_815 : Bool;
      HELP_OPERATOR_816 : Bool;
      HELP_OPERATOR_817 : Bool;
      HELP_OPERATOR_818 : Bool;
      HELP_OPERATOR_819 : Bool;
      HELP_OPERATOR_820 : Bool;
      HELP_OPERATOR_821 : Bool;
      HELP_OPERATOR_822 : Bool;
      HELP_OPERATOR_823 : Bool;
      HELP_OPERATOR_824 : Bool;
      HELP_OPERATOR_825 : Bool;
      HELP_OPERATOR_826 : Bool;
      HELP_OPERATOR_827 : Bool;
      HELP_OPERATOR_828 : Bool;
      HELP_OPERATOR_829 : Bool;
      HELP_OPERATOR_830 : Bool;
      HELP_OPERATOR_831 : Bool;
      HELP_OPERATOR_832 : Bool;
      HELP_OPERATOR_833 : Bool;
      HELP_OPERATOR_834 : Bool;
      HELP_OPERATOR_835 : Bool;
      HELP_OPERATOR_836 : Bool;
      HELP_OPERATOR_837 : Bool;
      HELP_OPERATOR_838 : Bool;
      HELP_OPERATOR_839 : Bool;
      HELP_OPERATOR_840 : Bool;
      HELP_OPERATOR_841 : Bool;
      HELP_OPERATOR_842 : Bool;
      HELP_OPERATOR_843 : Bool;
      HELP_OPERATOR_844 : Bool;
      HELP_OPERATOR_845 : Bool;
      HELP_OPERATOR_846 : Bool;
      HELP_OPERATOR_847 : Bool;
      HELP_OPERATOR_848 : Bool;
      HELP_OPERATOR_849 : Bool;
      HELP_OPERATOR_850 : Bool;
      HELP_OPERATOR_851 : Bool;
      HELP_OPERATOR_852 : Bool;
      HELP_OPERATOR_853 : Bool;
      HELP_OPERATOR_854 : Bool;
      HELP_OPERATOR_855 : Bool;
      HELP_OPERATOR_856 : Bool;
      HELP_OPERATOR_857 : Bool;
      HELP_OPERATOR_858 : Bool;
      HELP_OPERATOR_859 : Bool;
      HELP_OPERATOR_860 : Bool;
      HELP_OPERATOR_861 : Bool;
      HELP_OPERATOR_862 : Bool;
      HELP_OPERATOR_863 : Bool;
      HELP_OPERATOR_864 : Bool;
      HELP_OPERATOR_865 : Bool;
      HELP_OPERATOR_866 : Bool;
      HELP_OPERATOR_867 : Bool;
      HELP_OPERATOR_868 : Bool;
      HELP_OPERATOR_869 : Bool;
      HELP_OPERATOR_870 : Bool;
      HELP_OPERATOR_871 : Bool;
      HELP_OPERATOR_872 : Bool;
      HELP_OPERATOR_873 : Bool;
      HELP_OPERATOR_874 : Bool;
      HELP_OPERATOR_875 : Bool;
      HELP_OPERATOR_876 : Bool;
      HELP_OPERATOR_877 : Bool;
      HELP_OPERATOR_878 : Bool;
      HELP_OPERATOR_879 : Bool;
      HELP_OPERATOR_880 : Bool;
      HELP_OPERATOR_881 : Bool;
      HELP_OPERATOR_882 : Bool;
      HELP_OPERATOR_883 : Bool;
      HELP_OPERATOR_884 : Bool;
      HELP_OPERATOR_885 : Bool;
      HELP_OPERATOR_886 : Bool;
      HELP_OPERATOR_887 : Bool;
      HELP_OPERATOR_888 : Bool;
      HELP_OPERATOR_889 : Bool;
      HELP_OPERATOR_890 : Bool;
      HELP_OPERATOR_891 : Bool;
      HELP_OPERATOR_892 : Bool;
      HELP_OPERATOR_893 : Bool;
      HELP_OPERATOR_894 : Bool;
      HELP_OPERATOR_895 : Bool;
      HELP_OPERATOR_896 : Bool;
      HELP_OPERATOR_897 : Bool;
      HELP_OPERATOR_898 : Bool;
      HELP_OPERATOR_899 : Bool;
      HELP_OPERATOR_900 : Bool;   // RETURN GANTRY TO OUT OF COLLISION POSITION
      HELP_OPERATOR_901 : Bool;   // REQUEST GANTRY TO OPEN SAFETY GATES
      HELP_OPERATOR_902 : Bool;
      HELP_OPERATOR_903 : Bool;
      HELP_OPERATOR_904 : Bool;   // EMPTY THE ROBOT CELL
      HELP_OPERATOR_905 : Bool;
      HELP_OPERATOR_906 : Bool;
      HELP_OPERATOR_907 : Bool;
      HELP_OPERATOR_908 : Bool;
      HELP_OPERATOR_909 : Bool;
      HELP_OPERATOR_910 : Bool;
      HELP_OPERATOR_911 : Bool;
      HELP_OPERATOR_912 : Bool;
      HELP_OPERATOR_913 : Bool;
      HELP_OPERATOR_914 : Bool;
      HELP_OPERATOR_915 : Bool;
      HELP_OPERATOR_916 : Bool;
      HELP_OPERATOR_917 : Bool;
      HELP_OPERATOR_918 : Bool;
      HELP_OPERATOR_919 : Bool;
      HELP_OPERATOR_920 : Bool;
      HELP_OPERATOR_921 : Bool;
      HELP_OPERATOR_922 : Bool;
      HELP_OPERATOR_923 : Bool;
      HELP_OPERATOR_924 : Bool;
      HELP_OPERATOR_925 : Bool;   // RETURN ROBOT TO OUT OF COLLISION POSITION
      HELP_OPERATOR_926 : Bool;   // REQUEST ROBOT TO OPEN SAFETY GATES
      HELP_OPERATOR_927 : Bool;
      HELP_OPERATOR_928 : Bool;
      HELP_OPERATOR_929 : Bool;
      HELP_OPERATOR_930 : Bool;
      HELP_OPERATOR_931 : Bool;
      HELP_OPERATOR_932 : Bool;
      HELP_OPERATOR_933 : Bool;
      HELP_OPERATOR_934 : Bool;
      HELP_OPERATOR_935 : Bool;
      HELP_OPERATOR_936 : Bool;
      HELP_OPERATOR_937 : Bool;
      HELP_OPERATOR_938 : Bool;
      HELP_OPERATOR_939 : Bool;
      HELP_OPERATOR_940 : Bool;
      HELP_OPERATOR_941 : Bool;
      HELP_OPERATOR_942 : Bool;
      HELP_OPERATOR_943 : Bool;
      HELP_OPERATOR_944 : Bool;
      HELP_OPERATOR_945 : Bool;
      HELP_OPERATOR_946 : Bool;
      HELP_OPERATOR_947 : Bool;
      HELP_OPERATOR_948 : Bool;
      HELP_OPERATOR_949 : Bool;
      HELP_OPERATOR_950 : Bool;
      HELP_OPERATOR_951 : Bool;
      HELP_OPERATOR_952 : Bool;
      HELP_OPERATOR_953 : Bool;
      HELP_OPERATOR_954 : Bool;
      HELP_OPERATOR_955 : Bool;
      HELP_OPERATOR_956 : Bool;
      HELP_OPERATOR_957 : Bool;
      HELP_OPERATOR_958 : Bool;
      HELP_OPERATOR_959 : Bool;
      HELP_OPERATOR_960 : Bool;
      HELP_OPERATOR_961 : Bool;
      HELP_OPERATOR_962 : Bool;
      HELP_OPERATOR_963 : Bool;
      HELP_OPERATOR_964 : Bool;
      HELP_OPERATOR_965 : Bool;
      HELP_OPERATOR_966 : Bool;
      HELP_OPERATOR_967 : Bool;
      HELP_OPERATOR_968 : Bool;
      HELP_OPERATOR_969 : Bool;
      HELP_OPERATOR_970 : Bool;
      HELP_OPERATOR_971 : Bool;
      HELP_OPERATOR_972 : Bool;
      HELP_OPERATOR_973 : Bool;
      HELP_OPERATOR_974 : Bool;
      HELP_OPERATOR_975 : Bool;
      HELP_OPERATOR_976 : Bool;
      HELP_OPERATOR_977 : Bool;
      HELP_OPERATOR_978 : Bool;
      HELP_OPERATOR_979 : Bool;
      HELP_OPERATOR_980 : Bool;
      HELP_OPERATOR_981 : Bool;
      HELP_OPERATOR_982 : Bool;
      HELP_OPERATOR_983 : Bool;
      HELP_OPERATOR_984 : Bool;
      HELP_OPERATOR_985 : Bool;
      HELP_OPERATOR_986 : Bool;
      HELP_OPERATOR_987 : Bool;
      HELP_OPERATOR_988 : Bool;
      HELP_OPERATOR_989 : Bool;
      HELP_OPERATOR_990 : Bool;
      HELP_OPERATOR_991 : Bool;
      HELP_OPERATOR_992 : Bool;
      HELP_OPERATOR_993 : Bool;
      HELP_OPERATOR_994 : Bool;
      HELP_OPERATOR_995 : Bool;
      HELP_OPERATOR_996 : Bool;
      HELP_OPERATOR_997 : Bool;
      HELP_OPERATOR_998 : Bool;
      HELP_OPERATOR_999 : Bool;
      HELP_OPERATOR_1000 : Bool;
   END_VAR
BEGIN
END_DATA_BLOCK
